	16#01000002:
		F_EtherCAT_VendorIDtoString := 'Beckhoff Automation GmbH & Co. KG';

	16#01000056:
		F_EtherCAT_VendorIDtoString := 'SICK AG';

	16#01000083:
		F_EtherCAT_VendorIDtoString := 'Omron Robotics and Safety Technologies, Inc.';

	16#01000089:
		F_EtherCAT_VendorIDtoString := 'Parker Hannifin Manufacturing S.r.l.';

	16#010000E8:
		F_EtherCAT_VendorIDtoString := 'Balluff GmbH';

	16#010000F9:
		F_EtherCAT_VendorIDtoString := 'Nidec ACIM Germany GmbH';

	16#010000FB:
		F_EtherCAT_VendorIDtoString := 'maxon precision motors, inc.';

	16#0100016A:
		F_EtherCAT_VendorIDtoString := 'Tsubakimoto Chain Co.';

	16#01000230:
		F_EtherCAT_VendorIDtoString := 'Weidmuller Interface (Shanghai) Co.,Ltd.';

	16#01000331:
		F_EtherCAT_VendorIDtoString := 'SHANGHAI SANY SCIENCE & TECHNOLOGY CO., LTD';

	16#0100034E:
		F_EtherCAT_VendorIDtoString := 'Infineon Technologies Americas Corp.';

	16#0100050C:
		F_EtherCAT_VendorIDtoString := 'ABB Engineering (Shanghai) Ltd.';

	16#01000604:
		F_EtherCAT_VendorIDtoString := 'Leica Geosystems AG';

	16#01000734:
		F_EtherCAT_VendorIDtoString := 'MULTIVAC Sepp Haggenmuller SE & Co. KG';

	16#01000766:
		F_EtherCAT_VendorIDtoString := 'Renesas Electronics Korea Co., Ltd.';

	16#010007D5:
		F_EtherCAT_VendorIDtoString := 'Bimba Manufacturing Company';

	16#010007EC:
		F_EtherCAT_VendorIDtoString := 'SCREEN Holdings Co., Ltd.';

	16#0100083E:
		F_EtherCAT_VendorIDtoString := 'Frencken America Inc.';

	16#01000844:
		F_EtherCAT_VendorIDtoString := 'KLA-Tencor Corporation';

	16#01000876:
		F_EtherCAT_VendorIDtoString := 'EDAC Electronics Technology (Hangzhou) Co., Ltd.';

	16#0100090C:
		F_EtherCAT_VendorIDtoString := 'CORE CORPORATION';

	16#0100091C:
		F_EtherCAT_VendorIDtoString := 'Drobak Unlimited Co.';

	16#01000E3C:
		F_EtherCAT_VendorIDtoString := 'ADM Automation Ltd.';

	16#01000E9E:
		F_EtherCAT_VendorIDtoString := 'Optotune Slovakia s.r.o.';

	16#01001946:
		F_EtherCAT_VendorIDtoString := 'AMADA MIYACHI EUROPE GmbH';

	16#01003610:
		F_EtherCAT_VendorIDtoString := 'eProLinkTek Co., Ltd.';

	16#01007170:
		F_EtherCAT_VendorIDtoString := 'Hyundai Heavy Industries Holdings Co. Ltd.';

	16#01007680:
		F_EtherCAT_VendorIDtoString := 'HUNAN SUPER INFORMATION CO., LTD';

	16#0100ADDA:
		F_EtherCAT_VendorIDtoString := 'Fraunhofer-Institut fur Lasertechnik (ILT)';

	16#01053258:
		F_EtherCAT_VendorIDtoString := 'Shenzhen Encom Electric Technologies Co., Ltd.';

	16#01681168:
		F_EtherCAT_VendorIDtoString := 'Kinco Electric (Shenzhen) Ltd.';

	16#012EBC73:
		F_EtherCAT_VendorIDtoString := 'TIME GROUP Inc.';

	16#01ABCDEF:
		F_EtherCAT_VendorIDtoString := 'Ma.Vi. s.r.l.';

	16#02000089:
		F_EtherCAT_VendorIDtoString := 'Parker Hannifin Manufacturing Germany GmbH & Co KG';

	16#0200008D:
		F_EtherCAT_VendorIDtoString := 'Danfoss Drives A/S';

	16#02000331:
		F_EtherCAT_VendorIDtoString := 'SHANGHAI SANY SCIENCE & TECHNOLOGY CO., LTD';

	16#0200034E:
		F_EtherCAT_VendorIDtoString := 'Infineon Technologies China Co., Ltd.';

	16#0200ADDA:
		F_EtherCAT_VendorIDtoString := 'Fraunhofer-Institut fur Lasertechnik (ILT)';

	16#0300008D:
		F_EtherCAT_VendorIDtoString := 'Danfoss S.r.l.';

	16#04000089:
		F_EtherCAT_VendorIDtoString := 'Parker Hannifin Ltd.';

	16#04210909:
		F_EtherCAT_VendorIDtoString := 'Longxin Zhijian Co. Ltd.';

	16#04533417:
		F_EtherCAT_VendorIDtoString := 'MEYSAR MAKINA ELEKTRONIK ENERJI YAZILIM SAN. TIC. LTD. STI';

	16#05000089:
		F_EtherCAT_VendorIDtoString := 'Parker Hannifin Corporation';

	16#0505ABCD:
		F_EtherCAT_VendorIDtoString := 'A.L.L. Lasersysteme GmbH';

	16#0512FDFD:
		F_EtherCAT_VendorIDtoString := 'Suzhou GFD Automation Technology Co., Ltd';

	16#06402200:
		F_EtherCAT_VendorIDtoString := 'L-3 Communications, Communication Systems - West';

	16#06958326:
		F_EtherCAT_VendorIDtoString := 'BNT';

	16#07770777:
		F_EtherCAT_VendorIDtoString := 'Japan Radio Co., Ltd.';

	16#0800005A:
		F_EtherCAT_VendorIDtoString := 'Schneider Electric SE';

	16#08000089:
		F_EtherCAT_VendorIDtoString := 'Parker Hannifin Manufacturing Germany GmbH & Co. KG';

	16#09000089:
		F_EtherCAT_VendorIDtoString := 'Parker Hannifin Corporation';

	16#0A5D0000:
		F_EtherCAT_VendorIDtoString := 'Advanced Systems Development BVBA';

	16#0ADAFFFF:
		F_EtherCAT_VendorIDtoString := 'DSP Automation';

	16#0C044BAC:
		F_EtherCAT_VendorIDtoString := 'Compac Sorting Equipment Ltd.';

	16#0FA00000:
		F_EtherCAT_VendorIDtoString := 'FASTECH Co., Ltd.';

	16#0FFF8888:
		F_EtherCAT_VendorIDtoString := 'GSK CNC EQUIPMENT CO., LTD.';

	16#10000000:
		F_EtherCAT_VendorIDtoString := 'SONOTRONIC Nagel GmbH';

	16#10000001:
		F_EtherCAT_VendorIDtoString := 'XI’AN MOSVO ELECTRONICS TECHNOLOGY CO.,LTD';

	16#10000004:
		F_EtherCAT_VendorIDtoString := 'ED Co., Ltd';

	16#10000031:
		F_EtherCAT_VendorIDtoString := 'SHANGHAI SANY SCIENCE & TECHNOLOGY CO., LTD';

	16#10000331:
		F_EtherCAT_VendorIDtoString := 'SHANGHAI SANY SCIENCE & TECHNOLOGY CO., LTD';

	16#12345678:
		F_EtherCAT_VendorIDtoString := 'GA Drilling, Ltd.';

	16#17072003:
		F_EtherCAT_VendorIDtoString := 'METTEM-Specautomatic Ltd.';

	16#19491001:
		F_EtherCAT_VendorIDtoString := 'Tsinghua University, Department of Electronic Engineering';

	16#19821130:
		F_EtherCAT_VendorIDtoString := 'Control Z Corporation';

	16#19861230:
		F_EtherCAT_VendorIDtoString := 'Shanghai Damon Logistics Technology Co.,LTD';

	16#1BA90762:
		F_EtherCAT_VendorIDtoString := 'iba AG';

	16#20041961:
		F_EtherCAT_VendorIDtoString := 'Hengstler GmbH';

	16#20422B4C:
		F_EtherCAT_VendorIDtoString := 'Lenord, Bauer & Co. GmbH';

	16#20494154:
		F_EtherCAT_VendorIDtoString := 'Universitat Bremen, Institut fur Automatisierungstechnik (IAT)';

	16#22222222:
		F_EtherCAT_VendorIDtoString := 'Shanghai Cohere Electronics Technology Co., Ltd.';

	16#23091861:
		F_EtherCAT_VendorIDtoString := 'Robert Bosch GmbH';

	16#26262626:
		F_EtherCAT_VendorIDtoString := 'APDISAR (Association pour la Promotion et le Developpement de l’Ecole D’Ingenieurs ESISAR)';

	16#26376345:
		F_EtherCAT_VendorIDtoString := 'Convex Co., Ltd.';

	16#2E000000:
		F_EtherCAT_VendorIDtoString := 'X2E GmbH';

	16#30000331:
		F_EtherCAT_VendorIDtoString := 'SHANGHAI SANY SCIENCE & TECHNOLOGY CO., LTD';

	16#31313131:
		F_EtherCAT_VendorIDtoString := 'Sany Intelligent Control Equipment';

	16#31393633:
		F_EtherCAT_VendorIDtoString := 'Technische Universitat Darmstadt, Institut fur Elektromechanische Konstruktionen';

	16#314D4B54:
		F_EtherCAT_VendorIDtoString := 'MKT Systemtechnik GmbH & Co. KG';

	16#33333333:
		F_EtherCAT_VendorIDtoString := 'The ITAYA Engineering Ltd.';

	16#35409865:
		F_EtherCAT_VendorIDtoString := 'Korea Electronics Technology Institute';

	16#40000331:
		F_EtherCAT_VendorIDtoString := 'SHANGHAI SANY SCIENCE & TECHNOLOGY CO., LTD';

	16#40524F54:
		F_EtherCAT_VendorIDtoString := 'REDONE TECHNOLOGIES';

	16#414D4154:
		F_EtherCAT_VendorIDtoString := 'Applied Materials Inc.';

	16#41524341:
		F_EtherCAT_VendorIDtoString := 'ARCA TECNOLOGIE srl';

	16#4156414C:
		F_EtherCAT_VendorIDtoString := 'AVAL DATA CORPORATION';

	16#42000000:
		F_EtherCAT_VendorIDtoString := 'Trust Automation Inc.';

	16#43544C42:
		F_EtherCAT_VendorIDtoString := 'Central South University of Forestry and Technology, College of Computer Science and Information Technology';

	16#44454B31:
		F_EtherCAT_VendorIDtoString := 'DEK Printing Machines Ltd.';

	16#454C4F56:
		F_EtherCAT_VendorIDtoString := 'ELOVIS GmbH';

	16#454D5245:
		F_EtherCAT_VendorIDtoString := 'EKTECH Elektronik';

	16#46485320:
		F_EtherCAT_VendorIDtoString := 'SHF Communication Technologies AG';

	16#464D5331:
		F_EtherCAT_VendorIDtoString := 'FMS (Flexible Manufacturing System)';

	16#474F5353:
		F_EtherCAT_VendorIDtoString := 'Marcus Goner SYSTEM SOLUTIONS';

	16#47535953:
		F_EtherCAT_VendorIDtoString := 'Grossenbacher Systeme AG';

	16#482A0000:
		F_EtherCAT_VendorIDtoString := 'Hstar Technologies Corp.';

	16#48455673:
		F_EtherCAT_VendorIDtoString := 'University of Applied Sciences and Arts Western Switzerland (HES-SO - Valais Wallis), Institute of Systems Engineering';

	16#4C4E5449:
		F_EtherCAT_VendorIDtoString := 'NTI AG - LinMot';

	16#4C524358:
		F_EtherCAT_VendorIDtoString := 'Lam Research Corporation';

	16#4D4C5431:
		F_EtherCAT_VendorIDtoString := 'MLT Micro Laser Technology GmbH';

	16#50005000:
		F_EtherCAT_VendorIDtoString := 'Technische Universitat Braunschweig';

	16#50414E43:
		F_EtherCAT_VendorIDtoString := 'Power Automation GmbH';

	16#52414649:
		F_EtherCAT_VendorIDtoString := 'RAFI GmbH & Co. KG';

	16#53545A53:
		F_EtherCAT_VendorIDtoString := 'Steinbeis-Transferzentrum Systemtechnik';

	16#5445434E:
		F_EtherCAT_VendorIDtoString := 'Tecan Schweiz AG';

	16#54455753:
		F_EtherCAT_VendorIDtoString := 'TEWS Elektronik GmbH & Co. KG';

	16#54494158:
		F_EtherCAT_VendorIDtoString := 'Timax Electronics & Machinery Ltd.';

	16#55555555:
		F_EtherCAT_VendorIDtoString := 'OLYMPUS CORPORATION';

	16#5555AAAA:
		F_EtherCAT_VendorIDtoString := 'SIASUN Robot & Automation Co., Ltd.';

	16#55AA55AA:
		F_EtherCAT_VendorIDtoString := 'Green Field Control System (I) Pvt. Ltd.';

	16#55AA55BB:
		F_EtherCAT_VendorIDtoString := 'JT3, LLC';

	16#56475454:
		F_EtherCAT_VendorIDtoString := 'Volvo Group';

	16#6167656D:
		F_EtherCAT_VendorIDtoString := 'megatec electronic GmbH';

	16#65547241:
		F_EtherCAT_VendorIDtoString := 'Arte Motion S.p.A.';

	16#66666666:
		F_EtherCAT_VendorIDtoString := 'Chinese Academy of Sciences, Institute of Optics and Electronics (IOE)';

	16#66668888:
		F_EtherCAT_VendorIDtoString := 'Shenzhen Just Motion Control Electromechanics Co.,Ltd';

	16#7061756C:
		F_EtherCAT_VendorIDtoString := 'PAUL Maschinenfabrik GmbH & Co.KG';

	16#77776968:
		F_EtherCAT_VendorIDtoString := 'Mesacon Messelektronik GmbH Dresden';

	16#77778888:
		F_EtherCAT_VendorIDtoString := 'Shanghai Tech Full Electric Co., Ltd.';

	16#81696189:
		F_EtherCAT_VendorIDtoString := 'Shandong University, School of Electrical Engineering';

	16#88888888:
		F_EtherCAT_VendorIDtoString := 'ScandiNova Systems AB';

	16#89898989:
		F_EtherCAT_VendorIDtoString := 'Woojin Plaimm Co., Ltd';

	16#90646350:
		F_EtherCAT_VendorIDtoString := 'ROBOCUBETECH Co., Ltd';

	16#99998888:
		F_EtherCAT_VendorIDtoString := 'Shanghai STEP Electric Corporation';

	16#AAAA5555:
		F_EtherCAT_VendorIDtoString := 'Sunin Technology Inc.';

	16#AAAAAAAA:
		F_EtherCAT_VendorIDtoString := 'COMIZOA Co., Ltd.';

	16#AAAABBBB:
		F_EtherCAT_VendorIDtoString := 'OOO Ruchservomotor';

	16#AAAAFFFF:
		F_EtherCAT_VendorIDtoString := 'Dalian Jafeng Electronics Co., Ltd.';

	16#ADD1DA7A:
		F_EtherCAT_VendorIDtoString := 'ADDI-DATA GmbH';

	16#B0500001:
		F_EtherCAT_VendorIDtoString := 'Husky Injection Molding Systems Ltd.';

	16#BCDA0001:
		F_EtherCAT_VendorIDtoString := 'JINOID CO., LTD.';

	16#BE78EC01:
		F_EtherCAT_VendorIDtoString := 'Bertec Corporation';

	16#C0DECAFE:
		F_EtherCAT_VendorIDtoString := 'Analog Devices, Inc.';

	16#D4C3B2A1:
		F_EtherCAT_VendorIDtoString := 'PULOON Technology Inc.';

	16#DEADBEEF:
		F_EtherCAT_VendorIDtoString := 'Albert Handtmann Maschinenfabrik GmbH & Co. KG';

	16#DEBE50F7:
		F_EtherCAT_VendorIDtoString := 'Dewesoft d.o.o.';

ELSE
	F_EtherCAT_VendorIDtoString := 'No ID Matches.'; (*Last Update : Apr 08,2025*)
END_CASE

END_FUNCTION

// Interface/I_SafetyBase
INTERFACE I_SafetyBase EXTENDS I_BaseFB

PROPERTY DependenceFB : I_BaseFB
GET
END_GET
SET
END_SET
END_PROPERTY

PROPERTY OK : BOOL
GET
END_GET
END_PROPERTY

PROPERTY SafetyReset : I_SafetyReset
SET
END_SET
END_PROPERTY

END_INTERFACE

// Interface/I_SafetyReset
INTERFACE I_SafetyReset EXTENDS I_CyclicFB

METHOD Execute
VAR_INPUT
END_VAR
END_METHOD

PROPERTY PulseDuration : TIME
SET
END_SET
END_PROPERTY

END_INTERFACE

// Interface/I_SafetySimulation
INTERFACE I_SafetySimulation EXTENDS I_SafetyBase

METHOD SimulateSafetyDiag
VAR_INPUT
	SimulationValueDiag : UINT;
END_VAR
END_METHOD

METHOD SimulateSafetyState
VAR_INPUT
	SimulationValueState : USINT;
END_VAR
END_METHOD

END_INTERFACE

// Project Information/F_GetCompany
// This function has been automatically generated from the project information.
{attribute 'signature_flag' := '1073741824'}
{attribute 'TcGenerated'}
{attribute 'no-analysis'}
FUNCTION F_GetCompany : WSTRING
VAR_INPUT
	
END_VAR

F_GetCompany := "Beckhoff Automation LLC";

END_FUNCTION

// Project Information/F_GetTitle
// This function has been automatically generated from the project information.
{attribute 'signature_flag' := '1073741824'}
{attribute 'TcGenerated'}
{attribute 'no-analysis'}
FUNCTION F_GetTitle : WSTRING
VAR_INPUT
	
END_VAR

F_GetTitle := "SPT Diagnostic";

END_FUNCTION

// Project Information/F_GetVersion
// This function has been automatically generated from the project information.
{attribute 'signature_flag' := '1073741824'}
{attribute 'TcGenerated'}
{attribute 'no-analysis'}
FUNCTION F_GetVersion : ST_LibVersion
VAR_INPUT
	
END_VAR

F_GetVersion.iMajor := 3;
F_GetVersion.iMinor := 9;
F_GetVersion.iBuild := 0;
F_GetVersion.iRevision := 0;
F_GetVersion.sVersion := '3.9.0';
F_GetVersion.nFlags := 1;

END_FUNCTION

// Safety/Safety FBs Diagnostic/Reset Functionblocks/FB_SafetyResetPulse
FUNCTION_BLOCK FB_SafetyResetPulse EXTENDS FB_CyclicFB IMPLEMENTS I_SafetyReset
VAR
	// Reset Bit to connecto to Safety
	Reset AT %Q* : BOOL;

	// Internal Variables
	TpErrorAck	: TP;
	TofErrorAck : TOF;

	// Properties
	_PulseDuration : TIME := T#100MS;
END_VAR

METHOD CyclicLogic
IF NOT _InitComplete THEN
	_InitComplete := TRUE;
	RETURN;
END_IF

// Reset Logic
TpErrorAck(PT := _PulseDuration, Q => Reset);
IF TpErrorAck.Q THEN
	TpErrorAck.IN := FALSE;
END_IF

TofErrorAck(In := TpErrorAck.Q, PT := _PulseDuration); // Block Error messages for raising and falling edge of reset signal

// Status 
_Error	 := FALSE;
_ErrorId := 0;
_Busy	 := TofErrorAck.Q;
END_METHOD

METHOD Execute
IF TpErrorAck.Q THEN
	RETURN;
END_IF

TpErrorAck.IN := TRUE;
END_METHOD

PROPERTY PulseDuration : TIME
SET
_PulseDuration := PulseDuration;
END_SET
END_PROPERTY

END_FUNCTION_BLOCK

// Safety/Safety FBs Diagnostic/FB_Component_Safety_AndOrFB
{attribute 'no_explicit_call' := 'do not call this POU directly'}
FUNCTION_BLOCK FB_Component_Safety_AndOrFB EXTENDS FB_Component_Safety_Base

// This method serves as the entry point for all underlying FB logic
METHOD PUBLIC CyclicLogic

// This method should be called cyclically by descendant function blocks by invoking SUPER^.CyclicLogic().  Alternatively, the contents of this method could be reimplemented entirely in which case a call to this method would not be necessary.
IF NOT _InitComplete THEN
	_InitComplete := Initialize();
	RETURN;
END_IF

(* Main Component Signals*)
_OK		 := SUPER^.InfoData.State = E_ComponentSafetyOrAnd_State.Run;
_Busy	 := FALSE;
_ErrorId := 0;
SUPER^.CyclicLogic();
END_METHOD

// Basic component initialization logic
METHOD PROTECTED Initialize : BOOL;

// This method is called by CyclicLogic() as required
Initialize := SUPER^.Initialize();
END_METHOD

END_FUNCTION_BLOCK

// Safety/Safety FBs Diagnostic/FB_Component_Safety_Base
{attribute 'no_explicit_call' := 'do not call this POU directly'}
FUNCTION_BLOCK ABSTRACT FB_Component_Safety_Base EXTENDS FB_ComponentBase IMPLEMENTS I_SafetyBase, I_SafetySimulation
VAR
	InfoData AT %I* : ST_SafetyStateDiag;

	// Reset
	ipSafetyReset : I_SafetyReset;

	// Safety Status
	ipDependenceFB : I_BaseFB; // Pointer to FB this FB is dependent on
	_OK			   : BOOL;
END_VAR

// Clears error flags and error IDs for this component
METHOD PUBLIC Reset : BOOL
_Error	 := FALSE;
_ErrorId := 0;
IF ipSafetyReset <> 0 THEN
	ipSafetyReset.Execute();
END_IF

Reset := SUPER^.Reset();
END_METHOD

// This method serves as the entry point for all underlying FB logic
METHOD PUBLIC CyclicLogic

// This method should be called cyclically by descendant function blocks by invoking SUPER^.CyclicLogic().  Alternatively, the contents of this method could be reimplemented entirely in which case a call to this method would not be necessary.
IF NOT _InitComplete THEN
	_InitComplete := Initialize();
	RETURN;
END_IF

IF ipSafetyReset <> 0 THEN
	ipSafetyReset.CyclicLogic();
END_IF

SUPER^.CyclicLogic();
END_METHOD

PROPERTY DependenceFB : I_BaseFB
GET
DependenceFB := ipDependenceFB;
END_GET
SET
ipDependenceFB := DependenceFB;
END_SET
END_PROPERTY

{attribute 'monitoring' := 'variable'}
PROPERTY OK : BOOL
GET
OK := _OK;
END_GET
END_PROPERTY

PROPERTY SafetyReset : I_SafetyReset
SET
ipSafetyReset := SafetyReset;
END_SET
END_PROPERTY

METHOD SimulateSafetyDiag
VAR_INPUT
	SimulationValueDiag : UINT;
END_VAR
Infodata.Diag := SimulationValueDiag;
END_METHOD

METHOD SimulateSafetyState
VAR_INPUT
	SimulationValueState : USINT;
END_VAR
Infodata.State := SimulationValueState;
END_METHOD

// Basic component initialization logic
METHOD PROTECTED Initialize : BOOL;
{analysis -22}
IF NOT _Simulate THEN
	IF NOT _Error AND (F_GetMappingStatus(ADR(InfoData), SIZEOF(InfoData)) = EplcMappingStatus.MS_Unmapped) AND NOT _Simulate THEN
		_Error := TRUE;
		TRACE('Init Failed - State not mapped to Safety!');
	END_IF

	IF _Error THEN
		RETURN;
	END_IF
END_IF

Initialize := SUPER^.Initialize();
END_METHOD

END_FUNCTION_BLOCK

// Safety/Safety FBs Diagnostic/FB_Component_Safety_ConnectionFB
{attribute 'no_explicit_call' := 'do not call this POU directly'}
FUNCTION_BLOCK FB_Component_Safety_ConnectionFB EXTENDS FB_Component_Safety_Base
VAR
	// Alarms
	ComponentSafetyConnectionAlarms : ARRAY[1..COMPONENT_SAFETY_CONNECTION_ALARM_COUNT] OF FB_TcAlarm;
END_VAR

VAR CONSTANT
	COMPONENT_SAFETY_CONNECTION_ALARM_COUNT : UDINT := 20;
END_VAR

METHOD PROTECTED CreateEvents
VAR
END_VAR

// This method is called by Initialize() as required
F_CreateAllEventsInClass(Alarms		:= ComponentSafetyConnectionAlarms,
						 ClassSize	:= SIZEOF(TC_EVENTS.SafetyConnection),
						 pInitEvent := ADR(TC_EVENTS.SafetyConnection.InitReferenceEvent),
						 Prefix		:= Name);

SUPER^.CreateEvents();
END_METHOD

// Provides basic error detection and event handling for this component
METHOD PROTECTED Monitoring
VAR_INST
	DiagWord	: WORD;
	BitMaskDiag : WORD := 16#000F;
END_VAR

// This method is called cyclically by CyclicLogic()
SUPER^.Monitoring();
IF ipSafetyReset <> 0 AND_THEN ipSafetyReset.Busy THEN
	RETURN;
END_IF

BitMaskDiag := 16#000F;
DiagWord	:= TO_WORD(SUPER^.InfoData.Diag) AND BitMaskDiag;
IF (DiagWord = 1) AND NOT ComponentSafetyConnectionAlarms[E_SafetyConnection.InvalidCommand].bRaised THEN
	RaiseAlarmWithStrings(ComponentSafetyConnectionAlarms[E_SafetyConnection.InvalidCommand], '', '');
ELSIF NOT (DiagWord = 1) AND ComponentSafetyConnectionAlarms[E_SafetyConnection.InvalidCommand].bRaised THEN
	ComponentSafetyConnectionAlarms[E_SafetyConnection.InvalidCommand].Clear(0, 0);
END_IF

IF (DiagWord = 2) AND NOT ComponentSafetyConnectionAlarms[E_SafetyConnection.UnknownCommand].bRaised THEN
	RaiseAlarmWithStrings(ComponentSafetyConnectionAlarms[E_SafetyConnection.UnknownCommand], '', '');
ELSIF NOT (DiagWord = 2) AND ComponentSafetyConnectionAlarms[E_SafetyConnection.UnknownCommand].bRaised THEN
	ComponentSafetyConnectionAlarms[E_SafetyConnection.UnknownCommand].Clear(0, 0);
END_IF

IF (DiagWord = 3) AND NOT ComponentSafetyConnectionAlarms[E_SafetyConnection.InvalidConID].bRaised THEN
	RaiseAlarmWithStrings(ComponentSafetyConnectionAlarms[E_SafetyConnection.InvalidConID], '', '');
ELSIF NOT (DiagWord = 3) AND ComponentSafetyConnectionAlarms[E_SafetyConnection.InvalidConID].bRaised THEN
	ComponentSafetyConnectionAlarms[E_SafetyConnection.InvalidConID].Clear(0, 0);
END_IF

IF (DiagWord = 4) AND NOT ComponentSafetyConnectionAlarms[E_SafetyConnection.InvalidCrc].bRaised THEN
	RaiseAlarmWithStrings(ComponentSafetyConnectionAlarms[E_SafetyConnection.InvalidCrc], '', '');
ELSIF NOT (DiagWord = 4) AND ComponentSafetyConnectionAlarms[E_SafetyConnection.InvalidCrc].bRaised THEN
	ComponentSafetyConnectionAlarms[E_SafetyConnection.InvalidCrc].Clear(0, 0);
END_IF

IF (DiagWord = 5) AND NOT ComponentSafetyConnectionAlarms[E_SafetyConnection.WatchdogExpired].bRaised THEN
	RaiseAlarmWithStrings(ComponentSafetyConnectionAlarms[E_SafetyConnection.WatchdogExpired], '', '');
ELSIF NOT (DiagWord = 5) AND ComponentSafetyConnectionAlarms[E_SafetyConnection.WatchdogExpired].bRaised THEN
	ComponentSafetyConnectionAlarms[E_SafetyConnection.WatchdogExpired].Clear(0, 0);
END_IF

IF (DiagWord = 6) AND NOT ComponentSafetyConnectionAlarms[E_SafetyConnection.InvalidFSOEAddr].bRaised THEN
	RaiseAlarmWithStrings(ComponentSafetyConnectionAlarms[E_SafetyConnection.InvalidFSOEAddr], '', '');
ELSIF NOT (DiagWord = 6) AND ComponentSafetyConnectionAlarms[E_SafetyConnection.InvalidFSOEAddr].bRaised THEN
	ComponentSafetyConnectionAlarms[E_SafetyConnection.InvalidFSOEAddr].Clear(0, 0);
END_IF

IF (DiagWord = 7) AND NOT ComponentSafetyConnectionAlarms[E_SafetyConnection.InvalidData].bRaised THEN
	RaiseAlarmWithStrings(ComponentSafetyConnectionAlarms[E_SafetyConnection.InvalidData], '', '');
ELSIF NOT (DiagWord = 7) AND ComponentSafetyConnectionAlarms[E_SafetyConnection.InvalidData].bRaised THEN
	ComponentSafetyConnectionAlarms[E_SafetyConnection.InvalidData].Clear(0, 0);
END_IF

IF (DiagWord = 8) AND NOT ComponentSafetyConnectionAlarms[E_SafetyConnection.InvalidComParameterLen].bRaised THEN
	RaiseAlarmWithStrings(ComponentSafetyConnectionAlarms[E_SafetyConnection.InvalidComParameterLen], '', '');
ELSIF NOT (DiagWord = 8) AND ComponentSafetyConnectionAlarms[E_SafetyConnection.InvalidComParameterLen].bRaised THEN
	ComponentSafetyConnectionAlarms[E_SafetyConnection.InvalidComParameterLen].Clear(0, 0);
END_IF

IF (DiagWord = 9) AND NOT ComponentSafetyConnectionAlarms[E_SafetyConnection.InavlidComParameter].bRaised THEN
	RaiseAlarmWithStrings(ComponentSafetyConnectionAlarms[E_SafetyConnection.InavlidComParameter], '', '');
ELSIF NOT (DiagWord = 9) AND ComponentSafetyConnectionAlarms[E_SafetyConnection.InavlidComParameter].bRaised THEN
	ComponentSafetyConnectionAlarms[E_SafetyConnection.InavlidComParameter].Clear(0, 0);
END_IF

IF (DiagWord = 10) AND NOT ComponentSafetyConnectionAlarms[E_SafetyConnection.InvalidUserParameterLen].bRaised THEN
	RaiseAlarmWithStrings(ComponentSafetyConnectionAlarms[E_SafetyConnection.InvalidUserParameterLen], '', '');
ELSIF NOT (DiagWord = 10) AND ComponentSafetyConnectionAlarms[E_SafetyConnection.InvalidUserParameterLen].bRaised THEN
	ComponentSafetyConnectionAlarms[E_SafetyConnection.InvalidUserParameterLen].Clear(0, 0);
END_IF

IF (DiagWord = 11) AND NOT ComponentSafetyConnectionAlarms[E_SafetyConnection.InvalidUserParameter].bRaised THEN
	RaiseAlarmWithStrings(ComponentSafetyConnectionAlarms[E_SafetyConnection.InvalidUserParameter], '', '');
ELSIF NOT (DiagWord = 11) AND ComponentSafetyConnectionAlarms[E_SafetyConnection.InvalidUserParameter].bRaised THEN
	ComponentSafetyConnectionAlarms[E_SafetyConnection.InvalidUserParameter].Clear(0, 0);
END_IF

IF (DiagWord = 12) AND NOT ComponentSafetyConnectionAlarms[E_SafetyConnection.FSoEMasterReset].bRaised THEN
	RaiseAlarmWithStrings(ComponentSafetyConnectionAlarms[E_SafetyConnection.FSoEMasterReset], '', '');
ELSIF NOT (DiagWord = 12) AND ComponentSafetyConnectionAlarms[E_SafetyConnection.FSoEMasterReset].bRaised THEN
	ComponentSafetyConnectionAlarms[E_SafetyConnection.FSoEMasterReset].Clear(0, 0);
END_IF

IF (DiagWord = 13) AND NOT ComponentSafetyConnectionAlarms[E_SafetyConnection.ModuleErrorOnSlave].bRaised THEN
	RaiseAlarmWithStrings(ComponentSafetyConnectionAlarms[E_SafetyConnection.ModuleErrorOnSlave], '', '');
ELSIF NOT (DiagWord = 13) AND ComponentSafetyConnectionAlarms[E_SafetyConnection.ModuleErrorOnSlave].bRaised THEN
	ComponentSafetyConnectionAlarms[E_SafetyConnection.ModuleErrorOnSlave].Clear(0, 0);
END_IF

IF (DiagWord = 14) AND NOT ComponentSafetyConnectionAlarms[E_SafetyConnection.ModuleError].bRaised THEN
	RaiseAlarmWithStrings(ComponentSafetyConnectionAlarms[E_SafetyConnection.ModuleError], '', '');
ELSIF NOT (DiagWord = 14) AND ComponentSafetyConnectionAlarms[E_SafetyConnection.ModuleError].bRaised THEN
	ComponentSafetyConnectionAlarms[E_SafetyConnection.ModuleError].Clear(0, 0);
END_IF

IF (DiagWord = 15) AND NOT ComponentSafetyConnectionAlarms[E_SafetyConnection.SlaveNotStarted].bRaised THEN
	RaiseAlarmWithStrings(ComponentSafetyConnectionAlarms[E_SafetyConnection.SlaveNotStarted], '', '');
ELSIF NOT (DiagWord = 15) AND ComponentSafetyConnectionAlarms[E_SafetyConnection.SlaveNotStarted].bRaised THEN
	ComponentSafetyConnectionAlarms[E_SafetyConnection.SlaveNotStarted].Clear(0, 0);
END_IF

BitMaskDiag := 16#0010;
DiagWord	:= TO_WORD(SUPER^.InfoData.Diag) AND BitMaskDiag;
IF DiagWord.4 AND NOT ComponentSafetyConnectionAlarms[E_SafetyConnection.FsoESlaveError].bRaised THEN
	RaiseAlarmWithStrings(ComponentSafetyConnectionAlarms[E_SafetyConnection.FsoESlaveError], '', '');
ELSIF NOT DiagWord.4 AND ComponentSafetyConnectionAlarms[E_SafetyConnection.FsoESlaveError].bRaised THEN
	ComponentSafetyConnectionAlarms[E_SafetyConnection.FsoESlaveError].Clear(0, 0);
END_IF

BitMaskDiag := 16#0020;
DiagWord	:= TO_WORD(SUPER^.InfoData.Diag) AND BitMaskDiag;
IF DiagWord.5 AND NOT ComponentSafetyConnectionAlarms[E_SafetyConnection.FsoESlaveFailSafeValue].bRaised THEN
	RaiseAlarmWithStrings(ComponentSafetyConnectionAlarms[E_SafetyConnection.FsoESlaveFailSafeValue], '', '');
ELSIF NOT DiagWord.5 AND ComponentSafetyConnectionAlarms[E_SafetyConnection.FsoESlaveFailSafeValue].bRaised THEN
	ComponentSafetyConnectionAlarms[E_SafetyConnection.FsoESlaveFailSafeValue].Clear(0, 0);
END_IF

BitMaskDiag := 16#0040;
DiagWord	:= TO_WORD(SUPER^.InfoData.Diag) AND BitMaskDiag;
IF DiagWord.6 AND NOT ComponentSafetyConnectionAlarms[E_SafetyConnection.Startup].bRaised THEN
	RaiseAlarmWithStrings(ComponentSafetyConnectionAlarms[E_SafetyConnection.Startup], '', '');
ELSIF NOT DiagWord.6 AND ComponentSafetyConnectionAlarms[E_SafetyConnection.Startup].bRaised THEN
	ComponentSafetyConnectionAlarms[E_SafetyConnection.Startup].Clear(0, 0);
END_IF

BitMaskDiag := 16#0080;
DiagWord	:= TO_WORD(SUPER^.InfoData.Diag) AND BitMaskDiag;
IF DiagWord.7 AND NOT ComponentSafetyConnectionAlarms[E_SafetyConnection.FsoEMasterSafeValue].bRaised THEN
	RaiseAlarmWithStrings(ComponentSafetyConnectionAlarms[E_SafetyConnection.FsoEMasterSafeValue], '', '');
ELSIF NOT DiagWord.7 AND ComponentSafetyConnectionAlarms[E_SafetyConnection.FsoEMasterSafeValue].bRaised THEN
	ComponentSafetyConnectionAlarms[E_SafetyConnection.FsoEMasterSafeValue].Clear(0, 0);
END_IF

_CurrentAlarmSeverity := F_GetMaxSeverityRaised(Alarms := ComponentSafetyConnectionAlarms, CurrentSeverity := _CurrentAlarmSeverity);
END_METHOD

// Clears error flags and error IDs for this component
METHOD PUBLIC Reset : BOOL
F_ClearAllEventsInClass(ComponentSafetyConnectionAlarms);
Reset := SUPER^.Reset();
END_METHOD

// This method serves as the entry point for all underlying FB logic
METHOD PUBLIC CyclicLogic
// This method should be called cyclically by descendant function blocks by invoking SUPER^.CyclicLogic().  Alternatively, the contents of this method could be reimplemented entirely in which case a call to this method would not be necessary.
VAR
	i : UDINT;
END_VAR
IF NOT _InitComplete THEN
	_InitComplete := Initialize();
	RETURN;
END_IF

(* Main Component Signals*)
_OK		 := SUPER^.InfoData.State = E_ComponentSafetyConnection_State.Data;
_Busy	 := FALSE;
_ErrorId := SUPER^.InfoData.Diag;
SUPER^.CyclicLogic();
END_METHOD

// Basic component initialization logic
METHOD PROTECTED Initialize : BOOL;

// This method is called by CyclicLogic() as required
Initialize := SUPER^.Initialize();
END_METHOD

END_FUNCTION_BLOCK

// Safety/Safety FBs Diagnostic/FB_Component_Safety_EdmFB
{attribute 'no_explicit_call' := 'do not call this POU directly'}
FUNCTION_BLOCK FB_Component_Safety_EdmFB EXTENDS FB_Component_Safety_Base
VAR
	// Alarms
	ComponentSafetyEDMAlarms : ARRAY[1..COMPONENT_SAFETY_EDM_ALARM_COUNT] OF FB_TcAlarm;
END_VAR

VAR CONSTANT
	COMPONENT_SAFETY_EDM_ALARM_COUNT : UDINT := 3;
END_VAR

METHOD PROTECTED CreateEvents
VAR
END_VAR

// This method is called by Initialize() as required
F_CreateAllEventsInClass(Alarms		:= ComponentSafetyEdmAlarms,
						 ClassSize	:= SIZEOF(TC_EVENTS.SafetyEdm),
						 pInitEvent := ADR(TC_EVENTS.SafetyEdm.InitReferenceEvent),
						 Prefix		:= Name);

SUPER^.CreateEvents();
END_METHOD

// Provides basic error detection and event handling for this component
METHOD PROTECTED Monitoring

//This method is called cyclically by CyclicLogic()
SUPER^.Monitoring();

// No error evaluation if upper Level of Safety (Group or connection) is faulted  
IF ipDependenceFB <> 0 THEN
	IF ipDependenceFB.Error THEN
		F_ClearAllEventsInClass(ComponentSafetyEdmAlarms);
		RETURN;
	END_IF
END_IF

IF ipSafetyReset <> 0 AND_THEN ipSafetyReset.Busy THEN
	RETURN;
END_IF

IF SUPER^.InfoData.Diag.0 AND NOT ComponentSafetyEdmAlarms[E_SafetyEdm.SwitchOffTime].bRaised THEN
	RaiseAlarmWithStrings(ComponentSafetyEdmAlarms[E_SafetyEdm.SwitchOffTime], '', '');
ELSIF NOT SUPER^.InfoData.Diag.0 AND ComponentSafetyEdmAlarms[E_SafetyEdm.SwitchOffTime].bRaised THEN
	ComponentSafetyEdmAlarms[E_SafetyEdm.SwitchOffTime].Clear(0, 0);
END_IF

IF SUPER^.InfoData.Diag.1 AND NOT ComponentSafetyEdmAlarms[E_SafetyEdm.SwitchOnTime].bRaised THEN
	RaiseAlarmWithStrings(ComponentSafetyEdmAlarms[E_SafetyEdm.SwitchOnTime], '', '');
ELSIF NOT SUPER^.InfoData.Diag.1 AND ComponentSafetyEdmAlarms[E_SafetyEdm.SwitchOnTime].bRaised THEN
	ComponentSafetyEdmAlarms[E_SafetyEdm.SwitchOnTime].Clear(0, 0);
END_IF

_CurrentAlarmSeverity := F_GetMaxSeverityRaised(Alarms := ComponentSafetyEdmAlarms, CurrentSeverity := _CurrentAlarmSeverity);
END_METHOD

// Clears error flags and error IDs for this component
METHOD PUBLIC Reset : BOOL
F_ClearAllEventsInClass(ComponentSafetyEDMAlarms);
Reset := SUPER^.Reset();
END_METHOD

// This method serves as the entry point for all underlying FB logic
METHOD PUBLIC CyclicLogic
// This method should be called cyclically by descendant function blocks by invoking SUPER^.CyclicLogic().  Alternatively, the contents of this method could be reimplemented entirely in which case a call to this method would not be necessary.
VAR
	i : UDINT;
END_VAR
IF NOT _InitComplete THEN
	_InitComplete := Initialize();
	RETURN;
END_IF

(* Main Component Signals*)
_OK		 := SUPER^.InfoData.State <> E_ComponentSafetyEdm_State.Error;
_Busy	 := FALSE;
_ErrorId := SUPER^.InfoData.Diag;
SUPER^.CyclicLogic();
END_METHOD

// Basic component initialization logic
METHOD PROTECTED Initialize : BOOL;

// This method is called by CyclicLogic() as required
Initialize := SUPER^.Initialize();
END_METHOD

END_FUNCTION_BLOCK

// Safety/Safety FBs Diagnostic/FB_Component_Safety_EstopFB
{attribute 'no_explicit_call' := 'do not call this POU directly'}
FUNCTION_BLOCK FB_Component_Safety_EstopFB EXTENDS FB_Component_Safety_Base
VAR
	// Internal Variables
	_ActiveName : STRING := 'pressed!';

	// Alarms
	ComponentSafetyEstopAlarms : ARRAY[1..COMPONENT_SAFETY_ESTOP_ALARM_COUNT] OF FB_TcAlarm;
END_VAR

VAR CONSTANT
	COMPONENT_SAFETY_ESTOP_ALARM_COUNT : UDINT := 8;
END_VAR

METHOD PROTECTED CreateEvents
VAR
END_VAR

// This method is called by Initialize() as required
F_CreateAllEventsInClass(Alarms		:= ComponentSafetyEstopAlarms,
						 ClassSize	:= SIZEOF(TC_EVENTS.SafetyEstop),
						 pInitEvent := ADR(TC_EVENTS.SafetyEstop.InitReferenceEvent),
						 Prefix		:= Name);

SUPER^.CreateEvents();
END_METHOD

// Provides basic error detection and event handling for this component
METHOD PROTECTED Monitoring

//This method is called cyclically by CyclicLogic()
SUPER^.Monitoring();

// No error evaluation if upper Level of Safety (Group or connection) is faulted  
IF ipDependenceFB <> 0 THEN
	IF ipDependenceFB.Error THEN
		F_ClearAllEventsInClass(ComponentSafetyEstopAlarms);
		RETURN;
	END_IF
END_IF

IF ipSafetyReset <> 0 AND_THEN ipSafetyReset.Busy THEN
	RETURN;
END_IF

IF NOT SUPER^.OK AND NOT ComponentSafetyEstopAlarms[E_SafetyEstop.Active].bRaised THEN
	RaiseAlarmWithStrings(ComponentSafetyEstopAlarms[E_SafetyEstop.Active], _ActiveName, '');
ELSIF SUPER^.OK AND ComponentSafetyEstopAlarms[E_SafetyEstop.Active].bRaised THEN
	ComponentSafetyEstopAlarms[E_SafetyEstop.Active].Clear(0, 0);
END_IF

IF SUPER^.InfoData.Diag.0 AND NOT ComponentSafetyEstopAlarms[E_SafetyEstop.Disc1].bRaised THEN
	RaiseAlarmWithStrings(ComponentSafetyEstopAlarms[E_SafetyEstop.Disc1], '', '');
ELSIF NOT SUPER^.InfoData.Diag.0 AND ComponentSafetyEstopAlarms[E_SafetyEstop.Disc1].bRaised THEN
	ComponentSafetyEstopAlarms[E_SafetyEstop.Disc1].Clear(0, 0);
END_IF

IF SUPER^.InfoData.Diag.1 AND NOT ComponentSafetyEstopAlarms[E_SafetyEstop.Disc2].bRaised THEN
	RaiseAlarmWithStrings(ComponentSafetyEstopAlarms[E_SafetyEstop.Disc2], '', '');
ELSIF NOT SUPER^.InfoData.Diag.1 AND ComponentSafetyEstopAlarms[E_SafetyEstop.Disc2].bRaised THEN
	ComponentSafetyEstopAlarms[E_SafetyEstop.Disc2].Clear(0, 0);
END_IF

IF SUPER^.InfoData.Diag.2 AND NOT ComponentSafetyEstopAlarms[E_SafetyEstop.Disc3].bRaised THEN
	RaiseAlarmWithStrings(ComponentSafetyEstopAlarms[E_SafetyEstop.Disc3], '', '');
ELSIF NOT SUPER^.InfoData.Diag.2 AND ComponentSafetyEstopAlarms[E_SafetyEstop.Disc3].bRaised THEN
	ComponentSafetyEstopAlarms[E_SafetyEstop.Disc3].Clear(0, 0);
END_IF

IF SUPER^.InfoData.Diag.3 AND NOT ComponentSafetyEstopAlarms[E_SafetyEstop.Disc4].bRaised THEN
	RaiseAlarmWithStrings(ComponentSafetyEstopAlarms[E_SafetyEstop.Disc4], '', '');
ELSIF NOT SUPER^.InfoData.Diag.3 AND ComponentSafetyEstopAlarms[E_SafetyEstop.Disc4].bRaised THEN
	ComponentSafetyEstopAlarms[E_SafetyEstop.Disc4].Clear(0, 0);
END_IF

IF SUPER^.InfoData.Diag.4 AND NOT ComponentSafetyEstopAlarms[E_SafetyEstop.EDM1].bRaised THEN
	RaiseAlarmWithStrings(ComponentSafetyEstopAlarms[E_SafetyEstop.EDM1], '', '');
ELSIF NOT SUPER^.InfoData.Diag.4 AND ComponentSafetyEstopAlarms[E_SafetyEstop.EDM1].bRaised THEN
	ComponentSafetyEstopAlarms[E_SafetyEstop.EDM1].Clear(0, 0);
END_IF

IF SUPER^.InfoData.Diag.5 AND NOT ComponentSafetyEstopAlarms[E_SafetyEstop.EDM2].bRaised THEN
	RaiseAlarmWithStrings(ComponentSafetyEstopAlarms[E_SafetyEstop.EDM2], '', '');
ELSIF NOT SUPER^.InfoData.Diag.5 AND ComponentSafetyEstopAlarms[E_SafetyEstop.EDM2].bRaised THEN
	ComponentSafetyEstopAlarms[E_SafetyEstop.EDM2].Clear(0, 0);
END_IF

_CurrentAlarmSeverity := F_GetMaxSeverityRaised(Alarms := ComponentSafetyEstopAlarms, CurrentSeverity := _CurrentAlarmSeverity);
END_METHOD

// Clears error flags and error IDs for this component
METHOD PUBLIC Reset : BOOL
F_ClearAllEventsInClass(ComponentSafetyEstopAlarms);
Reset := SUPER^.Reset();
END_METHOD

// This method serves as the entry point for all underlying FB logic
METHOD PUBLIC CyclicLogic
// This method should be called cyclically by descendant function blocks by invoking SUPER^.CyclicLogic().  Alternatively, the contents of this method could be reimplemented entirely in which case a call to this method would not be necessary.
VAR
	i : UDINT;
END_VAR
IF NOT _InitComplete THEN
	_InitComplete := Initialize();
	RETURN;
END_IF

(* Main Component Signals*)
_OK		 := SUPER^.InfoData.State = E_ComponentSafetyEStop_State.Run;
_Busy	 := FALSE;
_ErrorId := SUPER^.InfoData.Diag;
SUPER^.CyclicLogic();
END_METHOD

PROPERTY ActiveName : STRING
SET
_ActiveName := ActiveName;
END_SET
END_PROPERTY

// Basic component initialization logic
METHOD PROTECTED Initialize : BOOL;

// This method is called by CyclicLogic() as required
Initialize := SUPER^.Initialize();
END_METHOD

END_FUNCTION_BLOCK

// Safety/Safety FBs Diagnostic/FB_Component_Safety_Group
{attribute 'no_explicit_call' := 'do not call this POU directly'}
FUNCTION_BLOCK FB_Component_Safety_Group EXTENDS FB_Component_Safety_Base
VAR
	// Safety Group Connections
	Run AT %Q* : BOOL;

	// Internal Variables
	AutoFaultAck	 : TON;
	TriggerAutoReset : R_TRIG;
	ConnectionError	 : BOOL;

	// Properties
	_AutoResetConnectionFaults : BOOL;

	// Alarms
	ComponentSafetyGroupAlarms : ARRAY[1..COMPONENT_SAFETY_GROUP_ALARM_COUNT] OF FB_TcAlarm;
END_VAR

VAR CONSTANT
	COMPONENT_SAFETY_GROUP_ALARM_COUNT : UDINT := 7;
END_VAR

METHOD PROTECTED CreateEvents
VAR
END_VAR

// This method is called by Initialize() as required
F_CreateAllEventsInClass(Alarms		:= ComponentSafetyGroupAlarms,
						 ClassSize	:= SIZEOF(TC_EVENTS.SafetyGroup),
						 pInitEvent := ADR(TC_EVENTS.SafetyGroup.InitReferenceEvent),
						 Prefix		:= Name);

SUPER^.CreateEvents();
END_METHOD

// Provides basic error detection and event handling for this component
METHOD PROTECTED Monitoring

//This method is called cyclically by CyclicLogic()
SUPER^.Monitoring();
IF ipSafetyReset <> 0 AND_THEN ipSafetyReset.Busy THEN
	RETURN;
END_IF

IF SUPER^.InfoData.Diag = E_ComponentSafetyGroup_Diag.FbError AND NOT ComponentSafetyGroupAlarms[E_SafetyGroup.FbError].bRaised THEN
	RaiseAlarmWithStrings(ComponentSafetyGroupAlarms[E_SafetyGroup.FbError], '', '');
ELSIF SUPER^.InfoData.Diag <> E_ComponentSafetyGroup_Diag.FbError AND ComponentSafetyGroupAlarms[E_SafetyGroup.FbError].bRaised THEN
	ComponentSafetyGroupAlarms[E_SafetyGroup.FbError].Clear(0, 0);
END_IF

IF SUPER^.InfoData.Diag = E_ComponentSafetyGroup_Diag.ComError AND NOT ComponentSafetyGroupAlarms[E_SafetyGroup.ComError].bRaised THEN
	RaiseAlarmWithStrings(ComponentSafetyGroupAlarms[E_SafetyGroup.ComError], '', '');
ELSIF SUPER^.InfoData.Diag <> E_ComponentSafetyGroup_Diag.ComError AND ComponentSafetyGroupAlarms[E_SafetyGroup.ComError].bRaised THEN
	ComponentSafetyGroupAlarms[E_SafetyGroup.ComError].Clear(0, 0);
END_IF

IF SUPER^.InfoData.Diag = E_ComponentSafetyGroup_Diag.ModuleError AND NOT ComponentSafetyGroupAlarms[E_SafetyGroup.ModuleError].bRaised THEN
	RaiseAlarmWithStrings(ComponentSafetyGroupAlarms[E_SafetyGroup.ModuleError], '', '');
ELSIF SUPER^.InfoData.Diag <> E_ComponentSafetyGroup_Diag.ModuleError AND ComponentSafetyGroupAlarms[E_SafetyGroup.ModuleError].bRaised THEN
	ComponentSafetyGroupAlarms[E_SafetyGroup.ModuleError].Clear(0, 0);
END_IF

IF SUPER^.InfoData.Diag = E_ComponentSafetyGroup_Diag.CmpError AND NOT ComponentSafetyGroupAlarms[E_SafetyGroup.CmpError].bRaised THEN
	RaiseAlarmWithStrings(ComponentSafetyGroupAlarms[E_SafetyGroup.CmpError], '', '');
ELSIF SUPER^.InfoData.Diag <> E_ComponentSafetyGroup_Diag.CmpError AND ComponentSafetyGroupAlarms[E_SafetyGroup.CmpError].bRaised THEN
	ComponentSafetyGroupAlarms[E_SafetyGroup.CmpError].Clear(0, 0);
END_IF

IF SUPER^.InfoData.Diag = E_ComponentSafetyGroup_Diag.DeactiveError AND NOT ComponentSafetyGroupAlarms[E_SafetyGroup.DeactiveError].bRaised THEN
	RaiseAlarmWithStrings(ComponentSafetyGroupAlarms[E_SafetyGroup.DeactiveError], '', '');
ELSIF SUPER^.InfoData.Diag <> E_ComponentSafetyGroup_Diag.DeactiveError AND ComponentSafetyGroupAlarms[E_SafetyGroup.DeactiveError].bRaised THEN
	ComponentSafetyGroupAlarms[E_SafetyGroup.DeactiveError].Clear(0, 0);
END_IF

IF SUPER^.InfoData.Diag = E_ComponentSafetyGroup_Diag.RestartError AND NOT ComponentSafetyGroupAlarms[E_SafetyGroup.RestartError].bRaised THEN
	RaiseAlarmWithStrings(ComponentSafetyGroupAlarms[E_SafetyGroup.RestartError], '', '');
ELSIF SUPER^.InfoData.Diag <> E_ComponentSafetyGroup_Diag.RestartError AND ComponentSafetyGroupAlarms[E_SafetyGroup.RestartError].bRaised THEN
	ComponentSafetyGroupAlarms[E_SafetyGroup.RestartError].Clear(0, 0);
END_IF

_CurrentAlarmSeverity := F_GetMaxSeverityRaised(Alarms := ComponentSafetyGroupAlarms, CurrentSeverity := _CurrentAlarmSeverity);
END_METHOD

// Clears error flags and error IDs for this component
METHOD PUBLIC Reset : BOOL
F_ClearAllEventsInClass(ComponentSafetyGroupAlarms);
Reset := SUPER^.Reset();
END_METHOD

// This method serves as the entry point for all underlying FB logic
METHOD PUBLIC CyclicLogic
// This method should be called cyclically by descendant function blocks by invoking SUPER^.CyclicLogic().  Alternatively, the contents of this method could be reimplemented entirely in which case a call to this method would not be necessary.
VAR
	i : UDINT;
END_VAR
IF NOT _InitComplete THEN
	_InitComplete := Initialize();
	RETURN;
END_IF

(*Control Group Group*)
Run				:= TRUE;
ConnectionError := SUPER^.InfoData.Diag <> 0;
IF ipSafetyReset <> 0 THEN
	AutoFaultAck(IN := (_AutoResetConnectionFaults AND ConnectionError) AND NOT ipSafetyReset.Busy, PT := T#250MS);
	TriggerAutoReset(CLK := AutoFaultAck.Q);
	IF TriggerAutoReset.Q THEN
		ipSafetyReset.Execute();
	END_IF
END_IF

(* Main Component Signals*)
_OK		 := SUPER^.InfoData.State = E_ComponentSafetyGroup_State.Run;
_Busy	 := FALSE;
_ErrorId := SUPER^.InfoData.Diag;
SUPER^.CyclicLogic();
END_METHOD

PROPERTY AutoResetConnectionFaults : BOOL
GET
AutoResetConnectionFaults := _AutoResetConnectionFaults;
END_GET
SET
_AutoResetConnectionFaults := AutoResetConnectionFaults;
END_SET
END_PROPERTY

// Basic component initialization logic
METHOD PROTECTED Initialize : BOOL;

// This method is called by CyclicLogic() as required
{analysis -22}
IF NOT _Simulate THEN
	IF NOT _Error AND (F_GetMappingStatus(ADR(Run), SIZEOF(Run)) = EplcMappingStatus.MS_Unmapped) THEN
		_Error := TRUE;
		Trace('Init Failed - Group Run not mapped to Safety!');
	END_IF

	IF NOT _Error AND ipSafetyReset = 0 THEN
		_Error := TRUE;
		Trace('Init Failed - Group requires Safety Reset FB Instance!');
	END_IF
END_IF

IF _Error THEN
	RETURN;
END_IF

Initialize := SUPER^.Initialize();
END_METHOD

END_FUNCTION_BLOCK

// Safety/Safety FBs Diagnostic/FB_Component_Safety_MonFB
{attribute 'no_explicit_call' := 'do not call this POU directly'}
FUNCTION_BLOCK FB_Component_Safety_MonFB EXTENDS FB_Component_Safety_Base
VAR
	// Alarm at Safe State
	_ActiveAlarm : BOOL	  := TRUE;
	_ActiveName	 : STRING := 'pressed!';

	// Alarms
	ComponentSafetyMonAlarms : ARRAY[1..COMPONENT_SAFETY_MON_ALARM_COUNT] OF FB_TcAlarm;
END_VAR

VAR CONSTANT
	COMPONENT_SAFETY_MON_ALARM_COUNT : UDINT := 10;
END_VAR

METHOD PROTECTED CreateEvents
VAR
END_VAR

// This method is called by Initialize() as required
F_CreateAllEventsInClass(Alarms		:= ComponentSafetyMonAlarms,
						 ClassSize	:= SIZEOF(TC_EVENTS.SafetyMon),
						 pInitEvent := ADR(TC_EVENTS.SafetyMon.InitReferenceEvent),
						 Prefix		:= Name);

SUPER^.CreateEvents();
END_METHOD

// Provides basic error detection and event handling for this component
METHOD PROTECTED Monitoring

// This method is called cyclically by CyclicLogic()
SUPER^.Monitoring();

// No error evaluation if upper Level of Safety (Group or connection) is faulted  
IF ipDependenceFB <> 0 THEN
	IF ipDependenceFB.Error THEN
		F_ClearAllEventsInClass(ComponentSafetyMonAlarms);
		RETURN;
	END_IF
END_IF

IF ipSafetyReset <> 0 AND_THEN ipSafetyReset.Busy THEN
	RETURN;
END_IF

IF NOT SUPER^.OK AND _ActiveAlarm AND NOT ComponentSafetyMonAlarms[E_SafetyMon.Active].bRaised THEN
	RaiseAlarmWithStrings(ComponentSafetyMonAlarms[E_SafetyMon.Active], _ActiveName, '');
ELSIF SUPER^.OK AND ComponentSafetyMonAlarms[E_SafetyMon.Active].bRaised THEN
	ComponentSafetyMonAlarms[E_SafetyMon.Active].Clear(0, 0);
END_IF

IF SUPER^.InfoData.Diag.0 AND NOT ComponentSafetyMonAlarms[E_SafetyMon.Disc1].bRaised THEN
	RaiseAlarmWithStrings(ComponentSafetyMonAlarms[E_SafetyMon.Disc1], '', '');
ELSIF NOT SUPER^.InfoData.Diag.0 AND ComponentSafetyMonAlarms[E_SafetyMon.Disc1].bRaised THEN
	ComponentSafetyMonAlarms[E_SafetyMon.Disc1].Clear(0, 0);
END_IF

IF SUPER^.InfoData.Diag.1 AND NOT ComponentSafetyMonAlarms[E_SafetyMon.Disc2].bRaised THEN
	RaiseAlarmWithStrings(ComponentSafetyMonAlarms[E_SafetyMon.Disc2], '', '');
ELSIF NOT SUPER^.InfoData.Diag.1 AND ComponentSafetyMonAlarms[E_SafetyMon.Disc2].bRaised THEN
	ComponentSafetyMonAlarms[E_SafetyMon.Disc2].Clear(0, 0);
END_IF

IF SUPER^.InfoData.Diag.3 AND NOT ComponentSafetyMonAlarms[E_SafetyMon.DiscInput].bRaised THEN
	RaiseAlarmWithStrings(ComponentSafetyMonAlarms[E_SafetyMon.DiscInput], '', '');
ELSIF NOT SUPER^.InfoData.Diag.3 AND ComponentSafetyMonAlarms[E_SafetyMon.DiscInput].bRaised THEN
	ComponentSafetyMonAlarms[E_SafetyMon.DiscInput].Clear(0, 0);
END_IF

IF SUPER^.InfoData.Diag.4 AND NOT ComponentSafetyMonAlarms[E_SafetyMon.Edm1].bRaised THEN
	RaiseAlarmWithStrings(ComponentSafetyMonAlarms[E_SafetyMon.Edm1], '', '');
ELSIF NOT SUPER^.InfoData.Diag.4 AND ComponentSafetyMonAlarms[E_SafetyMon.Edm1].bRaised THEN
	ComponentSafetyMonAlarms[E_SafetyMon.Edm1].Clear(0, 0);
END_IF

IF SUPER^.InfoData.Diag.5 AND NOT ComponentSafetyMonAlarms[E_SafetyMon.Edm2].bRaised THEN
	RaiseAlarmWithStrings(ComponentSafetyMonAlarms[E_SafetyMon.Edm2], '', '');
ELSIF NOT SUPER^.InfoData.Diag.5 AND ComponentSafetyMonAlarms[E_SafetyMon.Edm2].bRaised THEN
	ComponentSafetyMonAlarms[E_SafetyMon.Edm2].Clear(0, 0);
END_IF

IF SUPER^.InfoData.Diag.8 AND NOT ComponentSafetyMonAlarms[E_SafetyMon.Disc1Safe].bRaised THEN
	RaiseAlarmWithStrings(ComponentSafetyMonAlarms[E_SafetyMon.Disc1Safe], '', '');
ELSIF NOT SUPER^.InfoData.Diag.8 AND ComponentSafetyMonAlarms[E_SafetyMon.Disc1Safe].bRaised THEN
	ComponentSafetyMonAlarms[E_SafetyMon.Disc1Safe].Clear(0, 0);
END_IF

IF SUPER^.InfoData.Diag.9 AND NOT ComponentSafetyMonAlarms[E_SafetyMon.Disc2Safe].bRaised THEN
	RaiseAlarmWithStrings(ComponentSafetyMonAlarms[E_SafetyMon.Disc2Safe], '', '');
ELSIF NOT SUPER^.InfoData.Diag.9 AND ComponentSafetyMonAlarms[E_SafetyMon.Disc2Safe].bRaised THEN
	ComponentSafetyMonAlarms[E_SafetyMon.Disc2Safe].Clear(0, 0);
END_IF

IF SUPER^.InfoData.Diag.10 AND NOT ComponentSafetyMonAlarms[E_SafetyMon.DiscInputSafe].bRaised THEN
	RaiseAlarmWithStrings(ComponentSafetyMonAlarms[E_SafetyMon.DiscInputSafe], '', '');
ELSIF NOT SUPER^.InfoData.Diag.10 AND ComponentSafetyMonAlarms[E_SafetyMon.DiscInputSafe].bRaised THEN
	ComponentSafetyMonAlarms[E_SafetyMon.DiscInputSafe].Clear(0, 0);
END_IF

_CurrentAlarmSeverity := F_GetMaxSeverityRaised(Alarms := ComponentSafetyMonAlarms, CurrentSeverity := _CurrentAlarmSeverity);
END_METHOD

// Clears error flags and error IDs for this component
METHOD PUBLIC Reset : BOOL
F_ClearAllEventsInClass(ComponentSafetyMonAlarms);
Reset := SUPER^.Reset();
END_METHOD

// This method serves as the entry point for all underlying FB logic
METHOD PUBLIC CyclicLogic
// This method should be called cyclically by descendant function blocks by invoking SUPER^.CyclicLogic().  Alternatively, the contents of this method could be reimplemented entirely in which case a call to this method would not be necessary.
VAR
	i : UDINT;
END_VAR
IF NOT _InitComplete THEN
	_InitComplete := Initialize();
	RETURN;
END_IF

(* Main Component Signals*)
_OK		 := SUPER^.InfoData.State = E_ComponentSafetyMon_State.Run;
_Busy	 := FALSE;
_ErrorId := SUPER^.InfoData.Diag;
SUPER^.CyclicLogic();
END_METHOD

PROPERTY PUBLIC ActiveAlarm : BOOL
SET
_ActiveAlarm := ActiveAlarm;
END_SET
END_PROPERTY

PROPERTY ActiveName : STRING
SET
_ActiveName := ActiveName;
END_SET
END_PROPERTY

END_FUNCTION_BLOCK
